INTERFACE I_PressureSensor

METHOD getSignal : LREAL
VAR_INPUT
END_VAR
END_METHOD

METHOD setSignal : BOOL
VAR_INPUT
    input : LREAL;
END_VAR
END_METHOD

END_INTERFACE

(* stored: Version 1.1.0.1, ProductVersion 3.1.4024.9
   Itf I_PressureSensor: Id {3bf8359e-243c-41e8-8234-424e8868bde3}
   Method getSignal: Id {54d20a2a-1767-4441-a415-8d81638d9af3}
   Method setSignal: Id {e8d4b819-aa5c-4aa9-b64e-84daa4f8fee5} *)
